INTERFACE ITF_TopElement2_HMI_Connector EXTENDS ITF_BaseTopElement_HMI_Connector

END_INTERFACE

(* stored: Version 1.1.0.1, ProductVersion 3.1.4024.15
   Itf ITF_TopElement2_HMI_Connector: Id {61e297fe-6cc7-4777-8604-c349f66c2754} *)
